// TIA Portal V20 export
TYPE "LBP_typeModularMcpBaseOutput"
TITLE = Modular MCP image / Image MCP modulaire
// Output image of base signals for modular MCP / Image des sorties des signaux de base pour MCP modulaires
   STRUCT
      optionalKey1 : Bool;   // output image n+0 bit 0; KT-OUT1 / Image des sorties n+0 bit 0 ; KT-OUT1
      optionalKey2 : Bool;   // output image n+0 bit 1; KT-OUT2 / Image des sorties n+0 bit 1 ; KT-OUT2
      optionalKey3 : Bool;   // output image n+0 bit 2; KT-OUT3 / Image des sorties n+0 bit 2 ; KT-OUT3
      optionalKey4 : Bool;   // output image n+0 bit 3; KT-OUT4 / Image des sorties n+0 bit 3 ; KT-OUT4
      optionalKey5 : Bool;   // output image n+0 bit 4; KT-OUT5 / Image des sorties n+0 bit 4 ; KT-OUT5
      optionalKey6 : Bool;   // output image n+0 bit 5; KT-OUT6 / Image des sorties n+0 bit 5 ; KT-OUT6
      optionalKey7 : Bool;   // output image n+0 bit 6; KT-OUT7 / Image des sorties n+0 bit 6 ; KT-OUT7
      optionalKey8 : Bool;   // output image n+0 bit 7; KT-OUT8 / Image des sorties n+0 bit 7 ; KT-OUT8
      optionalKey9 : Bool;   // output image n+1 bit 0; KT-OUT9 / Image des sorties n+1 bit 0 ; KT-OUT9
      optionalKey10 : Bool;   // output image n+1 bit 1; KT-OUT10 / Image des sorties n+1 bit 1 ; KT-OUT10
      optionalKey11 : Bool;   // output image n+1 bit 2; KT-OUT11 / Image des sorties n+1 bit 2 ; KT-OUT11
      optionalKey12 : Bool;   // output image n+1 bit 3; KT-OUT12 / Image des sorties n+1 bit 3 ; KT-OUT12
      optionalKey13 : Bool;   // output image n+1 bit 4; KT-OUT13 / Image des sorties n+1 bit 4 ; KT-OUT13
      optionalKey14 : Bool;   // output image n+1 bit 5; KT-OUT14 / Image des sorties n+1 bit 5 ; KT-OUT14
      optionalKey15 : Bool;   // output image n+1 bit 6; KT-OUT15 / Image des sorties n+1 bit 6 ; KT-OUT15
      optionalKey16 : Bool;   // output image n+1 bit 7; KT-OUT16 / Image des sorties n+1 bit 7 ; KT-OUT16
   END_STRUCT;
END_TYPE
